Fanuc KAREL source: kb00047.KL

-- PROVISIONAL review KL for V1013-1; original PC SHA256 9049f11a1e0ab7bb80baca82b48827b3af1ed0ee0c63d9f49cefe7683f77cd0d
-- Incomplete behavior may be omitted. Consult companion uncertainty JSON. Do not deploy.
PROGRAM KB00047
%NOLOCKGROUP
BEGIN
  -- UNRESOLVED_PC offsets 5-14; opcodes 3F,75
  -- UNRESOLVED_PC offsets 19-28; opcodes 3F,75
  -- UNRESOLVED_PC offsets 33-40; opcodes 9D,23
  -- UNRESOLVED_PC offsets 45-52; opcodes 9D,23
  -- UNRESOLVED_PC offsets 57-89; opcodes 27,22,2A,22,2A,22,22,31
  -- UNRESOLVED_PC offsets 94-98; opcodes 7F
END KB00047
